# B&R Automation Studio project Tmp_Explorer_V1 (part 3)

#### USBdevice.st - Cyclic code
```iecst
PROGRAM _INIT
END_PROGRAM

PROGRAM _CYCLIC

	CASE state_machine OF
		// -----------------------------------------------------------------------------------------------------------
		// Wait state
		// -----------------------------------------------------------------------------------------------------------
		USB_WAIT:
			// Refresh USB data every X seconds when enabled
			node := 1;
			USB.status := ERR_OK;
			IF USB.CMD.auto_scan = TRUE THEN
				TON_10ms_01(IN:=1, PT:=USB.PAR.refresh_interval);
				// Get new USB data
				IF(TON_10ms_01.Q) THEN
					TON_10ms_01(IN:=0);
					USB.status := ERR_FUB_BUSY;
					brsmemset(ADR(usb_data), 0, SIZEOF(usb_data));
					state_machine := USB_CREATE_NODE_ID_LIST;
				END_IF
			ELSE
				TON_10ms_01(IN:=0);
			END_IF
			// Refresh USB data every X seconds when enabled
			IF USB.CMD.error_reset = TRUE THEN
				state_machine := USB_ERROR;
			END_IF
			// -----------------------------------------------------------------------------------------------------------
			// Get USB device list
			// -----------------------------------------------------------------------------------------------------------
		USB_CREATE_NODE_ID_LIST:
			UsbNodeListGet_0.enable := 1;
			UsbNodeListGet_0.pBuffer := ADR(node_id_buffer);
			UsbNodeListGet_0.bufferSize := SIZEOF(node_id_buffer);
			UsbNodeListGet_0.filterInterfaceClass := asusb_CLASS_MASS_STORAGE;
			UsbNodeListGet_0.filterInterfaceSubClass := 0;
			UsbNodeListGet_0;

			// --------------------------------------------------------------------------------------------------------------------
			// Success
			IF UsbNodeListGet_0.status = 0 THEN
				state_machine := USB_READ_DEVICE_DATA;
				node := 1;
				// No USB devices found
			ELSIF UsbNodeListGet_0.status = asusbERR_USB_NOTFOUND THEN
				// Unlink old device if it is gone now otherwise wait for next round
				FOR idx:=1 TO USB_MAX_CNT DO
					IF(USB.PAR.is_connected[idx] = TRUE) THEN
						node := 1;
						state_machine := USB_CHECK_LINKED;
						RETURN;
					END_IF
				END_FOR;
				state_machine := USB_WAIT;
				// Error
			ELSIF UsbNodeListGet_0.status <> ERR_FUB_BUSY THEN
				USB.status := UsbNodeListGet_0.status;
				USB.ERR.state := state_machine;
				IF UsbNodeListGet_0.status = asusbERR_BUFSIZE THEN
					USB.ERR.text := 'maximum number of devices reached';
				ELSE
					USB.ERR.text := 'error getting device list';
				END_IF;
				state_machine := USB_ERROR;
			END_IF;
			// -----------------------------------------------------------------------------------------------------------
			// Get device information
			// -----------------------------------------------------------------------------------------------------------
		USB_READ_DEVICE_DATA:
			UsbNodeGet_0.enable := 1;
			UsbNodeGet_0.nodeId := node_id_buffer[node];
			UsbNodeGet_0.pBuffer := ADR(usb_data[node]);
			UsbNodeGet_0.bufferSize := SIZEOF (usb_data[node]);
			UsbNodeGet_0;

			// --------------------------------------------------------------------------------------------------------------------
			// Success
			IF UsbNodeGet_0.status = 0 THEN
				// Make sure we have enough space to store USB data, proceed with next state_machine when all devices are detetced
				IF (node = UsbNodeListGet_0.listNodes) OR (node = USB_MAX_CNT) THEN
					node := 1;
					state_machine := USB_CHECK_LINKED;
					// Get next USB device
				ELSE
					node := node + 1;
				END_IF;
				// Error
			ELSIF UsbNodeGet_0.status <> ERR_FUB_BUSY THEN
				USB.status := UsbNodeGet_0.status;
				USB.ERR.state := state_machine;
				USB.ERR.text := 'error getting device data';
				state_machine := USB_ERROR;
			END_IF;
			// -----------------------------------------------------------------------------------------------------------
			// Check if linked device are still present
			// -----------------------------------------------------------------------------------------------------------
		USB_CHECK_LINKED:
			// Proceed to new devices when last device was checked
			IF(node > USB_MAX_CNT) THEN
				node := 1;
				state_machine := USB_LINK_NEW;
				RETURN;
			END_IF

			// -----------------------------------------------------------------------------------------------------------
			// Check if device is still active
			is_linked := FALSE;
			FOR idx:=1 TO USB_MAX_CNT DO
				// Compare old and new data
				IF(brsmemcmp(ADR(usb_data_old[node]), ADR(usb_data[idx]), SIZEOF(usb_data[idx])) = 0) AND
					(USB.PAR.ignore_dongle = FALSE OR (USB.PAR.ignore_dongle = TRUE AND usb_data[idx].productId <> BRproductId AND usb_data[idx].vendorId <> BRvendorId)) THEN
					// Clear data, mark as linked and EXIT loop
					brsmemset(ADR(usb_data[idx]), 0, SIZEOF(usb_data[idx]));
					is_linked := TRUE;
					EXIT;
				END_IF
			END_FOR;

			// -----------------------------------------------------------------------------------------------------------
			// Find next linked device
			IF(is_linked OR usb_data_old[node].interfaceClass = 0) THEN
				IF(node < USB_MAX_CNT) THEN
					node := node + 1;
					WHILE(node < USB_MAX_CNT AND usb_data_old[node].interfaceClass = 0) DO
						node := node + 1;
					END_WHILE;
					IF(node = USB_MAX_CNT AND usb_data_old[node].interfaceClass = 0) THEN
						node := node + 1;
					END_IF
				ELSE
					node := node + 1;
				END_IF
				// Unlink device if it is missing
			ELSE
				state_machine := USB_UNLINK_DEVICE;
			END_IF
			// -----------------------------------------------------------------------------------------------------------
			// Link new devices
			// -----------------------------------------------------------------------------------------------------------
		USB_LINK_NEW:
			// Return to wait state when last device was checked
			IF(node > USB_MAX_CNT) THEN
				state_machine := USB_WAIT;
				RETURN;
			END_IF

			// -----------------------------------------------------------------------------------------------------------
			// Find next new device
			IF(usb_data[node].interfaceClass <> 0) THEN
				IF(USB.PAR.ignore_dongle = FALSE OR (usb_data[node].productId <> BRproductId AND usb_data[node].vendorId <> BRvendorId)) THEN
					state_machine := USB_LINK_DEVICE;
					RETURN;
				END_IF
			END_IF
			node := node + 1;
			// -----------------------------------------------------------------------------------------------------------
			// Link device
			// -----------------------------------------------------------------------------------------------------------
		USB_LINK_DEVICE:
			// Find empty slot
			FOR idx:=1 TO USB_MAX_CNT DO
				IF(usb_data_old[idx].interfaceClass = 0) THEN
					EXIT;
				END_IF
			END_FOR;
			// No more slot available
			IF(idx = USB_MAX_CNT AND usb_data_old[idx].interfaceClass <> 0) THEN
				USB.status := ERR_MAX_DEVICE;
				USB.ERR.state := state_machine;
				USB.ERR.text := 'maximum number of device reached';
				state_machine := USB_ERROR;
				RETURN;
			END_IF
			// Create device string
			brsstrcpy(ADR(device_param), ADR('/DEVICE='));
			brsstrcat(ADR(device_param), ADR(usb_data[node].ifName));
			brsstrcpy(ADR(device_name), ADR('USB_DEVICE'));
			brsitoa(idx, ADR(tmpSTR));
			brsstrcat(ADR(device_name), ADR(tmpSTR));
			// Link device
			DevLink_0.enable := 1;
			DevLink_0.pDevice := ADR(device_name);
			DevLink_0.pParam := ADR(device_param);
			DevLink_0;

			// --------------------------------------------------------------------------------------------------------------------
			// Success
			IF DevLink_0.status = 0 THEN
				// Store data for new device
				brsmemcpy(ADR(usb_data_old[idx]), ADR(usb_data[node]), SIZEOF(usb_data[node]));
				USB.PAR.is_connected[idx] := TRUE;
				link_handle[idx] := DevLink_0.handle;
				node := node + 1;
				state_machine := USB_LINK_NEW;
				// Error
			ELSIF DevLink_0.status <> ERR_FUB_BUSY THEN
				USB.status := DevLink_0.status;
				USB.ERR.state := state_machine;
				USB.ERR.text := 'error linking device';
				state_machine := USB_ERROR;
			END_IF;
			// -----------------------------------------------------------------------------------------------------------
			// UnLink device
			// -----------------------------------------------------------------------------------------------------------
		USB_UNLINK_DEVICE:
			DevUnlink_0.enable := 1;
			DevUnlink_0.handle := link_handle[node];
			DevUnlink_0;

			// --------------------------------------------------------------------------------------------------------------------
			// Success
			IF DevUnlink_0.status = 0 THEN
				// Clear data
				brsmemset(ADR(usb_data_old[node]), 0, SIZEOF(usb_data_old[node]));
				USB.PAR.is_connected[node] := FALSE;
				link_handle[node] := 0;
				// Find next linked device
				WHILE(node < USB_MAX_CNT AND usb_data_old[node].interfaceClass = 0) DO
					node := node + 1;
				END_WHILE;
				IF(node = USB_MAX_CNT AND usb_data_old[node].interfaceClass = 0) THEN
					node := node + 1;
				END_IF
				state_machine := USB_CHECK_LINKED;
				// Error
			ELSIF DevUnlink_0.status <> ERR_FUB_BUSY THEN
				// Clear data
				brsmemset(ADR(usb_data_old[node]), 0, SIZEOF(usb_data_old[node]));
				USB.PAR.is_connected[node] := FALSE;
				link_handle[node] := 0;

				brsitoa(node, ADR(tmpSTR));
				USB.status := DevUnlink_0.status;
				USB.ERR.state := state_machine;
				USB.ERR.text := 'error unlinking device no ';
				brsstrcat(ADR(USB.ERR.text), ADR(tmpSTR));
				state_machine := USB_ERROR;
			END_IF;
			// -----------------------------------------------------------------------------------------------------------
			// Error state
			// -----------------------------------------------------------------------------------------------------------
		USB_ERROR:
			// Get more error information
			IF(USB.status = 0) THEN
				USB.status := FileIoGetSysError();
			END_IF

			// Unlink device
			IF(USB.ERR.state = USB_LINK_DEVICE) THEN
				DevUnlink_0.enable := 1;
				DevUnlink_0.handle := DevLink_0.handle;
				DevUnlink_0;
			END_IF

			// Reset error
			IF(USB.CMD.error_reset AND DevUnlink_0.status <> ERR_FUB_BUSY) THEN
				USB.CMD.error_reset := FALSE;
				brsmemset(ADR(USB.ERR), 0, SIZEOF(USB.ERR));
				state_machine := USB_WAIT;
			END_IF
	END_CASE;

END_PROGRAM

PROGRAM _EXIT
	FOR idx:=1 TO USB_MAX_CNT DO
		REPEAT
			DevUnlink_0.enable := 1;
			DevUnlink_0.handle := link_handle[idx];;
			DevUnlink_0;
			UNTIL DevUnlink_0.status <> ERR_FUB_BUSY
		END_REPEAT;
	END_FOR;
END_PROGRAM
```

#### USBdevice.var - Data for read_data Task
```iecst
(*----------------------------------------------------------------------------------------------------------------------------------------------------------------------------------------------------------------------------------------------------------------------*)
(*Local functions*)
VAR
	TON_10ms_01 : TON_10ms;
	UsbNodeListGet_0 : UsbNodeListGet; (*Type of FUB UsbNodeListGet*)
	UsbNodeGet_0 : UsbNodeGet; (*Type of FUB UsbNodeGet*)
	DevLink_0 : DevLink; (*Type of FUB DevLink*)
	DevUnlink_0 : DevUnlink; (*Type of FUB DevUnlink*)
END_VAR
(*----------------------------------------------------------------------------------------------------------------------------------------------------------------------------------------------------------------------------------------------------------------------*)
(*Local variables*)
VAR
	state_machine : usbSTATE; (*State machine*)
	device_param : STRING[80]; (*Connection path of USB device*)
	device_name : STRING[40]; (*Connection path of USB device*)
	link_handle : ARRAY[1..USB_MAX_CNT] OF UDINT; (*Link handle for USB device*)
	usb_data : ARRAY[1..USB_MAX_CNT] OF usbNode_typ; (*Data of all available USB devices*)
	usb_data_old : ARRAY[1..USB_MAX_CNT] OF usbNode_typ; (*Old data of all available USB devices*)
	node_id_buffer : ARRAY[1..USB_MAX_CNT] OF UDINT; (*Different nodeIDs saved in array-elements*)
	is_linked : BOOL; (*Helper variable that indicates that a USB stick is linked*)
	node : USINT; (*Node number*)
	idx : USINT;
	tmpSTR : STRING[10];
END_VAR
(*----------------------------------------------------------------------------------------------------------------------------------------------------------------------------------------------------------------------------------------------------------------------*)
(*Local constants*)
VAR CONSTANT
	BRvendorId : UINT := 1615; (*B&R vendor id*)
	BRproductId : UINT := 1001; (*B&R dongle product id*)
END_VAR
VAR
	ERR_MAX_DEVICE : UINT := 50000; (*Maximum number of dongles reached*)
END_VAR
```

### changelog.txt
```
Version 0.3
- Fixed USB reconnect issue

Version 0.2
- Support for multiple usb sticks

Version 0.1
- First public release
```

### NetTypes.typ
```iecst
TYPE
	netSTATE :
		(
		NET_WAIT, (*Function step: Wait for starting the Function chain*)
		NET_LINK_DEVICE, (*Function step: Link file device*)
		NET_UNLINK_DEVICE, (*Function step: Unlink the File Device from specific path*)
		NET_ERROR (*Function step: Jump to this step in every case of Error occuring in the Function chain*)
		);
	netCMD : 	STRUCT
		connect : BOOL := TRUE; (*Connect to network share*)
		disconnect : BOOL := TRUE; (*Disconnect from network share*)
		error_reset : BOOL; (*Reset error*)
	END_STRUCT;
	netPAR : 	STRUCT
		server_name : STRING[80]; (*Use server name*)
		server_ip : STRING[80] := '192.168.0.10'; (*or IP address*)
		server_port : STRING[80]; (*Uses default port when empty*)
		server_protocol : STRING[80] := 'cifs'; (*Type of network connection*)
		server_domain : STRING[80]; (*Domain name*)
		server_share : STRING[80] := 'share'; (*Name of the shared folder*)
		user_name : STRING[80] := 'user'; (*User name*)
		user_password : STRING[80] := 'password'; (*User password*)
		enable_connect : BOOL; (*Enable button connect*)
		can_ping : BOOL; (*Indicates that the network share can be pinged*)
		is_linked : BOOL; (*Network share is connected*)
	END_STRUCT;
	netERR : 	STRUCT
		state : netSTATE;
		text : STRING[80]; (*Error text*)
	END_STRUCT;
	netMAIN : 	STRUCT
		CMD : netCMD; (*Command structure*)
		PAR : netPAR; (*Parameter structure*)
		ERR : netERR; (*Error structure*)
		status : UINT;
	END_STRUCT;
END_TYPE
```

### NetVariables.var
```iecst
VAR
	PING_TIMEOUT : UINT := 200; (*Timeout for ping response*)
	NET : netMAIN;
END_VAR
```

### Program Logical/NETdevice/NetDevice (IEC)

#### Main.st - Init, cyclic, exit code
```iecst
PROGRAM _INIT
END_PROGRAM

PROGRAM _CYCLIC
	// Trigger ping request
	PingTimer.IN := TRUE;
	PingTimer.PT := PING_TIMEOUT;
	PingTimer();
	// Try to ping network share if not connected
	IF((NET.PAR.server_ip <> '' OR NET.PAR.server_name <> '') AND PingTimer.Q) THEN
		// Use IPÜ address
		IF(NET.PAR.server_ip <> '') THEN
			IcmpPing_0(enable := 1, pHost := ADR(NET.PAR.server_ip), timeout := PING_TIMEOUT);
		// Use host name
		ELSE
			IcmpPing_0(enable := 1, pHost := ADR(NET.PAR.server_name), timeout := PING_TIMEOUT);
		END_IF
		// Ping was OK
		IF(IcmpPing_0.status = ERR_OK) THEN
			PingTimer(IN := FALSE);
			NET.PAR.can_ping := TRUE;
		// Disconnect from share when ping failed
		ELSIF(IcmpPing_0.status <> ERR_FUB_BUSY) THEN
			PingTimer(IN := FALSE);
			NET.PAR.can_ping := FALSE;
			NET.CMD.disconnect := TRUE;
		END_IF
	ELSIF(PingTimer.Q) THEN
		PingTimer(IN := FALSE);
	END_IF

	CASE state_machine OF
		// -----------------------------------------------------------------------------------------------------------
		// Wait state
		// -----------------------------------------------------------------------------------------------------------
		NET_WAIT:
			NET.PAR.enable_connect := TRUE;
			NET.status := ERR_OK;
			// --------------------------------------------------------------------------------------------------------------------
			// Connect to server
			IF(NET.CMD.connect) THEN
				IF(NET.PAR.is_linked) THEN
					DevUnlink_0.enable := 0;
					DevUnlink_0;
					IF (DevUnlink_0.status = ERR_FUB_ENABLE_FALSE) THEN
						state_machine := NET_UNLINK_DEVICE;
					END_IF
				ELSE
					DevLink_0.enable := 0;
					DevLink_0;
					IF (DevLink_0.status = ERR_FUB_ENABLE_FALSE) THEN
						state_machine := NET_LINK_DEVICE;
					END_IF
				END_IF
				NET.status := ERR_FUB_BUSY;
			END_IF
			// --------------------------------------------------------------------------------------------------------------------
			// Disconnect from server
			IF(NET.CMD.disconnect) THEN
				IF(NET.PAR.is_linked) THEN
					DevUnlink_0.enable := 0;
					DevUnlink_0;
					state_machine := NET_UNLINK_DEVICE;
				ELSE
					NET.CMD.disconnect := FALSE;
				END_IF
			END_IF
			// --------------------------------------------------------------------------------------------------------------------
			// Reset error
			IF(NET.CMD.error_reset) THEN
				NET.CMD.error_reset := FALSE;
				brsmemset(ADR(NET.ERR), 0, SIZEOF(NET.ERR));
			END_IF
		// -----------------------------------------------------------------------------------------------------------
		// Link device
		// -----------------------------------------------------------------------------------------------------------
		NET_LINK_DEVICE:
			// Create device string
			NET.PAR.enable_connect := FALSE;
			brsmemset(ADR(device_param), 0, SIZEOF(device_param));
			IF(brsstrcmp(ADR(NET.PAR.server_name), ADR('')) <> 0) THEN
				brsstrcat(ADR(device_param), ADR('/SNAME='));
				brsstrcat(ADR(device_param), ADR(NET.PAR.server_name));
				brsstrcat(ADR(device_param), ADR(' '));
			END_IF
			IF(brsstrcmp(ADR(NET.PAR.server_ip), ADR('')) <> 0) THEN
				brsstrcat(ADR(device_param), ADR('/SIP='));
				brsstrcat(ADR(device_param), ADR(NET.PAR.server_ip));
				brsstrcat(ADR(device_param), ADR(' '));
			END_IF
			IF(brsstrcmp(ADR(NET.PAR.server_protocol), ADR('')) <> 0) THEN
				brsstrcat(ADR(device_param), ADR('/PROTOCOL='));
				brsstrcat(ADR(device_param), ADR(NET.PAR.server_protocol));
				brsstrcat(ADR(device_param), ADR(' '));
			END_IF
			IF(brsstrcmp(ADR(NET.PAR.server_port), ADR('')) <> 0) THEN
				brsstrcat(ADR(device_param), ADR('/PORT='));
				brsstrcat(ADR(device_param), ADR(NET.PAR.server_port));
				brsstrcat(ADR(device_param), ADR(' '));
			END_IF
			IF(brsstrcmp(ADR(NET.PAR.server_domain), ADR('')) <> 0) THEN
				brsstrcat(ADR(device_param), ADR('/DOMAIN='));
				brsstrcat(ADR(device_param), ADR(NET.PAR.server_domain));
				brsstrcat(ADR(device_param), ADR(' '));
			END_IF
			IF(brsstrcmp(ADR(NET.PAR.server_share), ADR('')) <> 0) THEN
				brsstrcat(ADR(device_param), ADR('/SHARE='));
				brsstrcat(ADR(device_param), ADR(NET.PAR.server_share));
				brsstrcat(ADR(device_param), ADR(' '));
			END_IF
			IF(brsstrcmp(ADR(NET.PAR.user_name), ADR('')) <> 0) THEN
				brsstrcat(ADR(device_param), ADR('/USER='));
				brsstrcat(ADR(device_param), ADR(NET.PAR.user_name));
				brsstrcat(ADR(device_param), ADR(' '));
			END_IF
			IF(brsstrcmp(ADR(NET.PAR.user_password), ADR('')) <> 0) THEN
				brsstrcat(ADR(device_param), ADR('/PASSWORD='));
				brsstrcat(ADR(device_param), ADR(NET.PAR.user_password));
				brsstrcat(ADR(device_param), ADR(' '));
			END_IF

			// Link device
			DevLink_0.enable := 1;
			DevLink_0.pDevice := ADR('NET_DEVICE');
			DevLink_0.pParam := ADR(device_param);
			DevLink_0;

			// --------------------------------------------------------------------------------------------------------------------
			// Success
			IF DevLink_0.status = 0 THEN
				device_handle := DevLink_0.handle;
				NET.PAR.is_linked := TRUE;
				NET.CMD.connect := FALSE;
				state_machine := NET_WAIT;
			// --------------------------------------------------------------------------------------------------------------------
			// Abort command
			ELSIF(NET.CMD.error_reset = TRUE OR NET.CMD.disconnect = TRUE) THEN
				NET.CMD.error_reset := FALSE;
				NET.CMD.connect := FALSE;
				state_machine := NET_WAIT;
			// Error
			ELSIF DevLink_0.status <> ERR_FUB_BUSY THEN
				NET.ERR.state := state_machine;
				NET.ERR.text := 'error linking device';
				NET.status := DevLink_0.status;
				state_machine := NET_ERROR;
			END_IF;
		// -----------------------------------------------------------------------------------------------------------
		// UnLink device
		// -----------------------------------------------------------------------------------------------------------
		NET_UNLINK_DEVICE:
			NET.PAR.enable_connect := FALSE;
			DevUnlink_0.enable := 1;
			DevUnlink_0.handle := device_handle;
			DevUnlink_0;

			// --------------------------------------------------------------------------------------------------------------------
			// Success
			IF DevUnlink_0.status = 0 THEN
				NET.PAR.is_linked := FALSE;
				IF(NET.CMD.connect) THEN
					DevLink_0.enable := 0;
					DevLink_0;
					state_machine := NET_LINK_DEVICE;
				ELSE
					NET.CMD.disconnect := FALSE;
					state_machine := NET_WAIT;
				END_IF
			// Error
			ELSIF DevUnlink_0.status <> ERR_FUB_BUSY THEN
				NET.CMD.error_reset := FALSE;
				NET.ERR.state := state_machine;
				NET.ERR.text := 'error unlinking device';
				NET.status := DevUnlink_0.status;
				state_machine := NET_ERROR;
			END_IF;
		// -----------------------------------------------------------------------------------------------------------
		// Error step
		// -----------------------------------------------------------------------------------------------------------
		NET_ERROR:
			// Reset commands
			NET.PAR.enable_connect := FALSE;
			NET.CMD.connect := FALSE;

			// Get more error information
			IF(NET.status = 0) THEN
				NET.status := FileIoGetSysError();
			END_IF
			IF(NET.status = 26228) THEN
				brsstrcpy(ADR(NET.ERR.text), ADR('connection rejected: check network protocol, username and password'));
			ELSIF(DevLink_0.status = fiERR_DEVICE_ALREADY_EXIST) THEN
				brsstrcpy(ADR(NET.ERR.text), ADR('device is already connected'));
			END_IF

			// Reset error
			IF(NET.CMD.error_reset) THEN
				NET.CMD.error_reset := FALSE;
				brsmemset(ADR(NET.ERR), 0, SIZEOF(NET.ERR));
				state_machine := NET_WAIT;
			END_IF
	END_CASE;

END_PROGRAM

PROGRAM _EXIT
	REPEAT
		DevUnlink_0.enable := 1;
		DevUnlink_0.handle := DevLink_0.handle;
		DevUnlink_0;
		UNTIL DevUnlink_0.status <> ERR_FUB_BUSY
	END_REPEAT;
END_PROGRAM
```

#### Variables.var - Local variables
```iecst
(*----------------------------------------------------------------------------------------------------------------------------------------------------------------------------------------------------------------------------------------------------------------------*)
(*Local functions*)
VAR
	DevLink_0 : DevLink; (*Link network device*)
	DevUnlink_0 : DevUnlink; (*Unlink network device*)
	IcmpPing_0 : IcmpPing; (*Ping network share*)
	PingTimer : TON_10ms;
END_VAR
(*----------------------------------------------------------------------------------------------------------------------------------------------------------------------------------------------------------------------------------------------------------------------*)
(*Local variables*)
VAR
	state_machine : netSTATE;
	device_param : STRING[200]; (*Connection path of network device*)
	device_handle : UDINT;
END_VAR
```

### changelog.txt
```
Version 0.3
- Remove state variable from PAR structure
- Added status variable to main structure
- Added disconnect command
- Ping is now executed all the time to detect connection interruption

Version 0.2
- Added ping support

Version 0.1
- First public release
```

Listed in the project but not available here: Logical/Global.typ, Logical/Global.var, Logical/Libraries/IecCheck/IecCheck.fun
